(* CoDeSys 2.3.9.55 project: ioBroker.modbus-codesys.pro *)
(* Libraries: Standard.lib 8.11.10 12:37:48, SYSLIBCALLBACK.LIB 8.11.10 12:37:48 *)

(* PLC configuration (modules and I/O channels)
K-Bus [K_Bus] node 0, in %IB0 out %QB0
Fieldbus variables [FB_VARS] node 1, in %IB0 out %QB0
Flag variables [FLAG_VARS] node 2, in %IB0 out %QB0
Modbus-Master [MB_MASTER] node 3, in %IB0 out %QB0
*)

(* Global variable list: Globale_Variablen *)
VAR_GLOBAL
	iob_read						AT %QW256:iob_read_t;
	iob_write						AT %MW128:iob_write_t;
END_VAR

(* Data type *)
TYPE iob_read_t :
STRUCT
	a_rd_BYTE:		BYTE;
	b_rd_WORD:		WORD;
	c_rd_DWORD:	DWORD;
	d_rd_SINT:		SINT;
	e_rd_INT:		INT;
	f_rd_UINT:		UINT;
	g_rd_DINT:		DINT;
	h_rd_UDINT:	UDINT;
	i_rd_REAL:		REAL;
	j_rd_STRING:	STRING;
	k_rd_TIME:		TIME;
	l_rd_TOD:		TOD;
	m_rd_DATE:		DATE;
	n_rd_DT:		DT;
	o_rd_ARRAY_INT: ARRAY[0..4] OF INT;
END_STRUCT
END_TYPE

(* Data type *)
TYPE iob_write_t :
STRUCT
	a_wr_BYTE:		BYTE;
	b_wr_WORD:		WORD;
	c_wr_DWORD:	DWORD;
	d_wr_SINT:		SINT;
	e_wr_INT:		INT;
	f_wr_UINT:		UINT;
	g_wr_DINT:		DINT;
	h_wr_UDINT:	UDINT;
	i_wr_REAL:		REAL;
	j_wr_STRING:	STRING;
	k_wr_TIME:		TIME;
	l_wr_TOD:		TOD;
	m_wr_DATE:		DATE;
	n_wr_DT:		DT;
	o_wr_ARRAY_INT: ARRAY[0..4] OF INT;
END_STRUCT
END_TYPE

(* POU PLC_PRG, ST *)
PROGRAM PLC_PRG
VAR
END_VAR
;
END_PROGRAM
